PROGRAM MAIN
VAR
	stMyTest : ST_Convert ;

END_VAR



PRG_PowerMeter() ;

PRG_Database();

END_PROGRAM

(* stored: Version 1.1.0.1, ProductVersion 3.1.4024.12
   POU MAIN: Id {b39c4d0b-2cf0-453e-b50b-5dbaaa464394}, SpecialFunc None *)
